PROGRAM PLC_AMX_AI
VAR_INPUT
	nSocketType:UINT:=1;// socket 类型; 0 表示 server; 1 表示 client;
	sTerminalName:STRING;// 通讯对方名称 自定义
	sHost:STRING(20):='127.0.0.1';// 通讯IP地址; server时表示本地host; client时表示远程host
	nPort:UDINT:=8900;// 通讯端口号;
	bEnable:BOOL:=TRUE;// 通讯启用\禁用连接
	sSendSuffix:STRING:='';//此处可统一添加发送后缀字符 $R$N
	nQueueInterval:UDINT:=50;// 发送队列时间间隔 单位ms
	logHandleArray:ARRAY [1..5] OF POINTER TO printLogModule_EX;// log 操作 handle 数组
	logHandleArrayLength:UINT:=0;// log 操作 handle 数组长度, 不超过5
	enHeartBeat:BOOL;// 启用心跳包命令
	cmdHeartBeat:DINT;// 心跳包命令
	readStateFlag:BOOL;
	volt:REAL;
	dworld:UDINT;
END_VAR
VAR_OUTPUT
	bSendCondition	:BOOL;//可发送条件
	bSocketConnected:BOOL;//连接状态
	
END_VAR
VAR CONSTANT
	cNumBegin		:DINT:=1;
	cNumEnd			:DINT:=100;
END_VAR
VAR
	sendDataArray	:ARRAY [cNumBegin..cNumEnd] OF struct_byte;
	length			:DINT:=0;
	endPoint		:DINT:=cNumBegin;
	sendPoint		:DINT:=cNumBegin;
	passMax			:BOOL;
	popupSendData	:struct_byte;
	//popup
	popupStep		:UINT:=0;
	popupTON1		:TON;
	popupTON2		:TON;
	iPopup			:DINT:=0;
	_PopupLength	:DINT:=0;
	sendDataTemp	:struct_byte;
	sendLenght		:UDINT;
END_VAR
VAR
	tcpipClient					:tcpipClientModule_EX;
	tcpipServer					:tcpipServerModule_EX;////定义服务器对象
	
	tcpipSendDataBuff_Server	:struct_byte;//发送数据 Buff server
	tcpipSendDataBuff_Client	:struct_byte;//发送数据 Buff client
	
	tcpipSendDataClear			:struct_byte;//发送数据 清空
	tcpipSendData				:struct_byte;//发送数据
	
	tcpipRecDataBuff_Server		:struct_byte;//已接收数据 Buff server
	tcpipRecDataBuff_Client		:struct_byte;//已接收数据 Buff client
	
	tcpipRecDataClear			:struct_byte;//已接收数据 清空
	tcpipRecData				:struct_byte;//已接收数据
	
	tcpConnectR_Trig			:R_Trig;//初始连接上升沿
	tcpConnectF_Trig			:F_Trig;//初始连接下降沿
	registerStep				:UDINT;//ALC注册控制步
	registerTON					:TON;//ALC注册延时
	
	logHandleArray_index		:UINT:=1;
	sendStep:UDINT;
	t1:TON;
	timeout1:TON;
	timeoutTimes:UDINT;
	disconnectedTon:TON;
END_VAR
VAR
	(*
	bTrig_Version:BOOL;
	rTrig_Version:R_TRIG;
	*)
END_VAR


CASE nSocketType OF
0://TCPIP server
	tcpipServer(
		sSrvNetId:= , 
		sLocalHost:=sHost , 
		nLocalPort:=nPort , 
		bStartConnect:=bEnable , 
		tcpipSDataLen:=sendLenght , 
		tcpipSData:=ADR(tcpipSendDataBuff_Server) , 
		bSend:= , 
		tcpipRecDataLen:=SIZEOF(tcpipRecDataBuff_Server), 
		tcpipRecData:=ADR(tcpipRecDataBuff_Server) , 
		bAccepted=> , 
		bSendBusy=> , 
		bRecData=> );
	bSendCondition:=tcpipServer.bAccepted AND NOT tcpipServer.bSendBusy;
	//TCPIP连接
	bSocketConnected:=tcpipServer.bAccepted;
	IF NOT tcpipServer.bAccepted THEN
		length:=0;
		endPoint:=cNumBegin;
		sendPoint:=cNumBegin;
		passMax:=FALSE;
	END_IF
	tcpConnectR_Trig(CLK:=tcpipServer.bAccepted);
	tcpConnectF_Trig(CLK:=tcpipServer.bAccepted);

1://TCPIP client
	tcpipClient(
		sSrvNetId:= , 
		sRemoteHost:=sHost , 
		nRemotePort:=nPort , 
		bStartConnect:=bEnable , 
		tcpipSDataLen:=sendLenght, 
		tcpipSData:=ADR(tcpipSendDataBuff_Client) , 
		bSend:= , 
		tcpipRecDataLen:=SIZEOF(tcpipRecDataBuff_Client) , 
		tcpipRecData:=ADR(tcpipRecDataBuff_Client) , 
		bConnected=> , 
		bSendBusy=> , 
		bRecData=> );
	bSendCondition:=tcpipClient.bConnected AND NOT tcpipClient.bSendBusy;
	//TCPIP连接
	bSocketConnected:=tcpipClient.bConnected;
	IF NOT tcpipClient.bConnected THEN
		length:=0;
		endPoint:=cNumBegin;
		sendPoint:=cNumBegin;
		passMax:=FALSE;
	END_IF
	tcpConnectR_Trig(CLK:=tcpipClient.bConnected);
	tcpConnectF_Trig(CLK:=tcpipClient.bConnected);
END_CASE

IF tcpConnectR_Trig.Q THEN
	FOR logHandleArray_index:=1 TO logHandleArrayLength DO
		logHandleArray[logHandleArray_index]^.append(CONCAT(sTerminalName, ' has been connected'));
	END_FOR
	registerStep:=10;
END_IF
IF tcpConnectF_Trig.Q THEN
	FOR logHandleArray_index:=1 TO logHandleArrayLength DO
		logHandleArray[logHandleArray_index]^.append(CONCAT(sTerminalName, ' has been disconnected'));
	END_FOR
	registerStep:=0;
END_IF
//数据接收处理
CASE nSocketType OF
0://TCPIP server
	IF tcpipServer.bRecData THEN
		tcpipRecData:=tcpipRecDataBuff_Server;//buff转存
		tcpipRecDataBuff_Server:=tcpipRecDataClear;//转存之后清空buff
		dataProcessing();
	END_IF
1://TCPIP client
	IF tcpipClient.bRecData THEN
		tcpipRecData:=tcpipRecDataBuff_Client;//buff转存
		tcpipRecDataBuff_Client:=tcpipRecDataClear;//转存之后清空buff
		dataProcessing();
	END_IF
END_CASE


popup();

CASE registerStep OF
0:
	//Ready
10:
	registerStep:=0;
// 心跳包
20:
	IF NOT enHeartBeat THEN
		registerStep:=0;
	ELSE
		registerStep:=registerStep+10;
	END_IF
30:
	registerTON(IN:=FALSE);
	registerStep:=registerStep+10;
40:
	registerTON(IN:=NOT registerTON.Q,PT:=T#3S);
	IF registerTON.Q THEN
		registerTON(IN:=FALSE);
		registerStep:=30;
	END_IF
END_CASE

CASE sendStep OF
0:
	sendStep:=10;
	timeout1(IN:=FALSE);
	t1(IN:=FALSE);
10:
	IF bSocketConnected THEN
		sendStep:=20;
	ELSE
		sendStep:=10;
	END_IF
// 心跳包
20:
	ReadVoltage();
	sendStep:=30;
30:
	IF readStateFlag THEN
		sendStep:=40;
		timeout1(IN:=FALSE);
		readStateFlag:=FALSE;
		timeoutTimes:=0;
		RETURN;
	END_IF
	timeout1(IN:=NOT timeout1.Q,PT:=T#1S);
	IF timeout1.Q THEN
		timeout1(IN:=FALSE);
		sendStep:=50;
		timeoutTimes:=timeoutTimes+1;
		IF timeoutTimes>3 THEN
			volt:=10.022;
			dworld:=4105;
			timeoutTimes:=0;
		END_IF
	END_IF
40:
	t1(IN:=NOT t1.Q,PT:=T#0.5S);
	IF t1.Q THEN
		t1(IN:=FALSE);
		sendStep:=50;
	END_IF
50:
	sendStep:=10;
END_CASE
disconnectedTon(IN:=NOT bSocketConnected,PT:=T#5S);
IF disconnectedTon.Q THEN
	volt:=10.022;
	dworld:=4105;
END_IF
Manual();

METHOD appendSend : BOOL
VAR_INPUT
	b1		:BYTE:=0;
	b2		:BYTE:=0;
	b3		:Byte:=0;
	b4		:Byte:=0;
	b5		:Byte:=0;
	b6		:Byte:=0;
	b7		:Byte:=0;
	b8		:Byte:=0;
	b9		:BYTE:=0;
	b10		:BYTE:=0;
	b11		:BYTE:=0;
	b12		:BYTE:=0;
	b13		:BYTE:=0;
	b14		:BYTE:=0;
	b15		:BYTE:=0;
	b16		:BYTE:=0;
	b17		:BYTE:=0;
	b18		:BYTE:=0;
	b19		:BYTE:=0;
	b20		:BYTE:=0;
	lenght	:UDINT;
END_VAR
sendLenght:=lenght;
sendDataArray[endPoint].b1:=b1;
sendDataArray[endPoint].b2:=b2;
sendDataArray[endPoint].b3:=b3;
sendDataArray[endPoint].b4:=b4;
sendDataArray[endPoint].b5:=b5;
sendDataArray[endPoint].b6:=b6;
sendDataArray[endPoint].b7:=b7;
sendDataArray[endPoint].b8:=b8;
sendDataArray[endPoint].b9:=b9;
sendDataArray[endPoint].b10:=b10;
sendDataArray[endPoint].b11:=b11;
sendDataArray[endPoint].b12:=b12;
sendDataArray[endPoint].b13:=b13;
sendDataArray[endPoint].b14:=b14;
sendDataArray[endPoint].b15:=b15;
sendDataArray[endPoint].b16:=b16;
sendDataArray[endPoint].b17:=b17;
sendDataArray[endPoint].b18:=b18;
sendDataArray[endPoint].b19:=b19;
sendDataArray[endPoint].b20:=b20;

endPoint:=endPoint+1;
IF endPoint>(cNumEnd-1) THEN
	endPoint:=1;
	passMax:=TRUE;
END_IF
END_METHOD

METHOD dataProcessing : BOOL
VAR_INPUT
END_VAR
VAR
	i_CGResult:INT;
	i_HResult:INT;
	str1:STRING;
END_VAR
FOR logHandleArray_index:=1 TO logHandleArrayLength DO
	CASE nSocketType OF
	0://TCPIP server
		str1:=CONCAT(str1,BYTE_TO_HEXSTR(tcpipRecData.b1,2,FALSE));
		str1:=CONCAT(str1,' ');
		str1:=CONCAT(str1,BYTE_TO_HEXSTR(tcpipRecData.b2,2,FALSE));
		str1:=CONCAT(str1,' ');
		str1:=CONCAT(str1,BYTE_TO_HEXSTR(tcpipRecData.b3,2,FALSE));
		str1:=CONCAT(str1,' ');
		str1:=CONCAT(str1,BYTE_TO_HEXSTR(tcpipRecData.b4,2,FALSE));
		str1:=CONCAT(str1,' ');
		str1:=CONCAT(str1,BYTE_TO_HEXSTR(tcpipRecData.b5,2,FALSE));
		str1:=CONCAT(str1,' ');
		str1:=CONCAT(str1,BYTE_TO_HEXSTR(tcpipRecData.b6,2,FALSE));
		str1:=CONCAT(str1,' ');
		str1:=CONCAT(str1,BYTE_TO_HEXSTR(tcpipRecData.b7,2,FALSE));
		str1:=CONCAT(str1,' ');
		str1:=CONCAT(str1,BYTE_TO_HEXSTR(tcpipRecData.b8,2,FALSE));
		str1:=CONCAT(str1,' ');
		str1:=CONCAT(str1,BYTE_TO_HEXSTR(tcpipRecData.b9,2,FALSE));
		str1:=CONCAT(str1,' ');
		str1:=CONCAT(str1,BYTE_TO_HEXSTR(tcpipRecData.b10,2,FALSE));
		str1:=CONCAT(str1,' ');
		str1:=CONCAT(str1,BYTE_TO_HEXSTR(tcpipRecData.b11,2,FALSE));
		str1:=CONCAT(str1,' ');
		str1:=CONCAT(str1,BYTE_TO_HEXSTR(tcpipRecData.b12,2,FALSE));
		str1:=CONCAT(str1,' ');
		str1:=CONCAT(str1,BYTE_TO_HEXSTR(tcpipRecData.b13,2,FALSE));
		str1:=CONCAT(str1,' ');
		str1:=CONCAT(str1,BYTE_TO_HEXSTR(tcpipRecData.b14,2,FALSE));
		str1:=CONCAT(str1,' ');
		str1:=CONCAT(str1,BYTE_TO_HEXSTR(tcpipRecData.b15,2,FALSE));
		str1:=CONCAT(str1,' ');
		str1:=CONCAT(str1,BYTE_TO_HEXSTR(tcpipRecData.b16,2,FALSE));
		str1:=CONCAT(str1,' ');
		str1:=CONCAT(str1,BYTE_TO_HEXSTR(tcpipRecData.b17,2,FALSE));
		str1:=CONCAT(str1,' ');
		str1:=CONCAT(str1,BYTE_TO_HEXSTR(tcpipRecData.b18,2,FALSE));
		str1:=CONCAT(str1,' ');
		str1:=CONCAT(str1,BYTE_TO_HEXSTR(tcpipRecData.b19,2,FALSE));
		str1:=CONCAT(str1,' ');
		str1:=CONCAT(str1,BYTE_TO_HEXSTR(tcpipRecData.b20,2,FALSE));
//		logHandleArray[logHandleArray_index]^.append(CONCAT(CONCAT(CONCAT('Recevie From ', sTerminalName), ' -- '),str1));
	1://TCPIP client
		str1:=CONCAT(str1,BYTE_TO_HEXSTR(tcpipRecData.b1,2,FALSE));
		str1:=CONCAT(str1,' ');
		str1:=CONCAT(str1,BYTE_TO_HEXSTR(tcpipRecData.b2,2,FALSE));
		str1:=CONCAT(str1,' ');
		str1:=CONCAT(str1,BYTE_TO_HEXSTR(tcpipRecData.b3,2,FALSE));
		str1:=CONCAT(str1,' ');
		str1:=CONCAT(str1,BYTE_TO_HEXSTR(tcpipRecData.b4,2,FALSE));
		str1:=CONCAT(str1,' ');
		str1:=CONCAT(str1,BYTE_TO_HEXSTR(tcpipRecData.b5,2,FALSE));
		str1:=CONCAT(str1,' ');
		str1:=CONCAT(str1,BYTE_TO_HEXSTR(tcpipRecData.b6,2,FALSE));
		str1:=CONCAT(str1,' ');
		str1:=CONCAT(str1,BYTE_TO_HEXSTR(tcpipRecData.b7,2,FALSE));
		str1:=CONCAT(str1,' ');
		str1:=CONCAT(str1,BYTE_TO_HEXSTR(tcpipRecData.b8,2,FALSE));
		str1:=CONCAT(str1,' ');
		str1:=CONCAT(str1,BYTE_TO_HEXSTR(tcpipRecData.b9,2,FALSE));
		str1:=CONCAT(str1,' ');
		str1:=CONCAT(str1,BYTE_TO_HEXSTR(tcpipRecData.b10,2,FALSE));
		str1:=CONCAT(str1,' ');
		str1:=CONCAT(str1,BYTE_TO_HEXSTR(tcpipRecData.b11,2,FALSE));
		str1:=CONCAT(str1,' ');
		str1:=CONCAT(str1,BYTE_TO_HEXSTR(tcpipRecData.b12,2,FALSE));
		str1:=CONCAT(str1,' ');
		str1:=CONCAT(str1,BYTE_TO_HEXSTR(tcpipRecData.b13,2,FALSE));
		str1:=CONCAT(str1,' ');
		str1:=CONCAT(str1,BYTE_TO_HEXSTR(tcpipRecData.b14,2,FALSE));
		str1:=CONCAT(str1,' ');
		str1:=CONCAT(str1,BYTE_TO_HEXSTR(tcpipRecData.b15,2,FALSE));
		str1:=CONCAT(str1,' ');
		str1:=CONCAT(str1,BYTE_TO_HEXSTR(tcpipRecData.b16,2,FALSE));
		str1:=CONCAT(str1,' ');
		str1:=CONCAT(str1,BYTE_TO_HEXSTR(tcpipRecData.b17,2,FALSE));
		str1:=CONCAT(str1,' ');
		str1:=CONCAT(str1,BYTE_TO_HEXSTR(tcpipRecData.b18,2,FALSE));
		str1:=CONCAT(str1,' ');
		str1:=CONCAT(str1,BYTE_TO_HEXSTR(tcpipRecData.b19,2,FALSE));
		str1:=CONCAT(str1,' ');
		str1:=CONCAT(str1,BYTE_TO_HEXSTR(tcpipRecData.b20,2,FALSE));
//		logHandleArray[logHandleArray_index]^.append(CONCAT(CONCAT(CONCAT('Recevie From ', sTerminalName), ' -- '),str1));
	END_CASE
END_FOR

// 数据处理
readStateFlag:=TRUE;
volt:=TO_REAL((tcpipRecData.b10*256+tcpipRecData.b11)/4096.0)*10.0;
dworld:=tcpipRecData.b10*256+tcpipRecData.b11;
END_METHOD

ACTION Manual:
(*
rTrig_Version(CLK:=bTrig_Version);
IF rTrig_Version.Q THEN
	appendSend(0,0,E_CmdID_SW.SW_GetVer,0.0,0.0,0.0,0.0,0.0,0,'');
END_IF
*)
END_ACTION

METHOD PRIVATE popup : BOOL
VAR_INPUT
END_VAR
CASE popupStep OF
0:
	IF (sendPoint<endPoint OR passMax) AND bSendCondition THEN
		popupSendData:=sendDataArray[sendPoint];
		sendData(popupSendData);//此处是调用信息发送
		popupStep:=10;
		sendPoint:=sendPoint+1;
		IF sendPoint>(cNumEnd-1) THEN
			sendPoint:=1;
			passMax:=FALSE;
		END_IF
	END_IF
10:
	popupTON2(IN:=NOT popupTON2.Q, PT:=T#2S);
	IF NOT bSendCondition OR popupTON2.Q THEN
		popupTON2(IN:=FALSE);
		popupStep:=11;
	END_IF
11:
	IF bSendCondition THEN
		popupStep:=12;
	END_IF
	popupTON1(IN:=FALSE);
12:
	//popupTON1(IN:=NOT popupTON1.Q,PT:=T#10MS);
	popupTON1(IN:=NOT popupTON1.Q,PT:=TO_TIME(nQueueInterval));
	IF popupTON1.Q THEN
		popupStep:=0;
	END_IF
END_CASE
END_METHOD

METHOD ReadVoltage : BOOL
VAR_INPUT
END_VAR
appendSend(16#00,16#00,16#00,16#00,16#00,16#06,16#01,16#04,16#00,16#00,16#00,16#04,0,0,0,0,0,0,0,0,12);// 读进电压字符串
END_METHOD

METHOD PRIVATE sendData : BOOL
VAR_INPUT
	dataStruct	:struct_byte;
END_VAR
VAR
	str1:STRING;
END_VAR
IF bSendCondition AND bEnable THEN
	tcpipSendData.b1	:=dataStruct.b1;
	tcpipSendData.b2	:=dataStruct.b2;
	tcpipSendData.b3	:=dataStruct.b3;
	tcpipSendData.b4	:=dataStruct.b4;
	tcpipSendData.b5	:=dataStruct.b5;
	tcpipSendData.b6	:=dataStruct.b6;
	tcpipSendData.b7	:=dataStruct.b7;
	tcpipSendData.b8	:=dataStruct.b8;
	tcpipSendData.b9	:=dataStruct.b9;
	tcpipSendData.b10	:=dataStruct.b10;
	tcpipSendData.b11	:=dataStruct.b11;
	tcpipSendData.b12	:=dataStruct.b12;
	tcpipSendData.b13	:=dataStruct.b13;
	tcpipSendData.b14	:=dataStruct.b14;
	tcpipSendData.b15	:=dataStruct.b15;
	tcpipSendData.b16	:=dataStruct.b16;
	tcpipSendData.b17	:=dataStruct.b17;
	tcpipSendData.b18	:=dataStruct.b18;
	tcpipSendData.b19	:=dataStruct.b19;
	tcpipSendData.b20	:=dataStruct.b20;
	
	CASE nSocketType OF
	0://TCPIP server
		tcpipSendDataBuff_Server:=tcpipSendData;
		tcpipSendData:=tcpipSendDataClear;	
		tcpipServer.bSend:=TRUE;
	1://TCPIP client
		tcpipSendDataBuff_Client:=tcpipSendData;
		tcpipSendData:=tcpipSendDataClear;	
		tcpipClient.bSend:=TRUE;
	END_CASE
	
	FOR logHandleArray_index:=1 TO logHandleArrayLength DO
		CASE nSocketType OF
		0://TCPIP server
			str1:=CONCAT(str1,BYTE_TO_HEXSTR(tcpipSendDataBuff_Server.b1,2,FALSE));
			str1:=CONCAT(str1,' ');
			str1:=CONCAT(str1,BYTE_TO_HEXSTR(tcpipSendDataBuff_Server.b2,2,FALSE));
			str1:=CONCAT(str1,' ');
			str1:=CONCAT(str1,BYTE_TO_HEXSTR(tcpipSendDataBuff_Server.b3,2,FALSE));
			str1:=CONCAT(str1,' ');
			str1:=CONCAT(str1,BYTE_TO_HEXSTR(tcpipSendDataBuff_Server.b4,2,FALSE));
			str1:=CONCAT(str1,' ');
			str1:=CONCAT(str1,BYTE_TO_HEXSTR(tcpipSendDataBuff_Server.b5,2,FALSE));
			str1:=CONCAT(str1,' ');
			str1:=CONCAT(str1,BYTE_TO_HEXSTR(tcpipSendDataBuff_Server.b6,2,FALSE));
			str1:=CONCAT(str1,' ');
			str1:=CONCAT(str1,BYTE_TO_HEXSTR(tcpipSendDataBuff_Server.b7,2,FALSE));
			str1:=CONCAT(str1,' ');
			str1:=CONCAT(str1,BYTE_TO_HEXSTR(tcpipSendDataBuff_Server.b8,2,FALSE));
			str1:=CONCAT(str1,' ');
			str1:=CONCAT(str1,BYTE_TO_HEXSTR(tcpipSendDataBuff_Server.b9,2,FALSE));
			str1:=CONCAT(str1,' ');
			str1:=CONCAT(str1,BYTE_TO_HEXSTR(tcpipSendDataBuff_Server.b10,2,FALSE));
			str1:=CONCAT(str1,' ');
			str1:=CONCAT(str1,BYTE_TO_HEXSTR(tcpipSendDataBuff_Server.b11,2,FALSE));
			str1:=CONCAT(str1,' ');
			str1:=CONCAT(str1,BYTE_TO_HEXSTR(tcpipSendDataBuff_Server.b12,2,FALSE));
			str1:=CONCAT(str1,' ');
			str1:=CONCAT(str1,BYTE_TO_HEXSTR(tcpipSendDataBuff_Server.b13,2,FALSE));
			str1:=CONCAT(str1,' ');
			str1:=CONCAT(str1,BYTE_TO_HEXSTR(tcpipSendDataBuff_Server.b14,2,FALSE));
			str1:=CONCAT(str1,' ');
			str1:=CONCAT(str1,BYTE_TO_HEXSTR(tcpipSendDataBuff_Server.b15,2,FALSE));
			str1:=CONCAT(str1,' ');
			str1:=CONCAT(str1,BYTE_TO_HEXSTR(tcpipSendDataBuff_Server.b16,2,FALSE));
			str1:=CONCAT(str1,' ');
			str1:=CONCAT(str1,BYTE_TO_HEXSTR(tcpipSendDataBuff_Server.b17,2,FALSE));
			str1:=CONCAT(str1,' ');
			str1:=CONCAT(str1,BYTE_TO_HEXSTR(tcpipSendDataBuff_Server.b18,2,FALSE));
			str1:=CONCAT(str1,' ');
			str1:=CONCAT(str1,BYTE_TO_HEXSTR(tcpipSendDataBuff_Server.b19,2,FALSE));
			str1:=CONCAT(str1,' ');
			str1:=CONCAT(str1,BYTE_TO_HEXSTR(tcpipSendDataBuff_Server.b20,2,FALSE));
//			logHandleArray[logHandleArray_index]^.append(CONCAT(CONCAT(CONCAT('Send To ', sTerminalName), ' -- '),str1));
		1://TCPIP client
			str1:=CONCAT(str1,' ');
			str1:=CONCAT(str1,BYTE_TO_HEXSTR(tcpipSendDataBuff_Client.b1,2,FALSE));
			str1:=CONCAT(str1,' ');
			str1:=CONCAT(str1,BYTE_TO_HEXSTR(tcpipSendDataBuff_Client.b2,2,FALSE));
			str1:=CONCAT(str1,' ');
			str1:=CONCAT(str1,BYTE_TO_HEXSTR(tcpipSendDataBuff_Client.b3,2,FALSE));
			str1:=CONCAT(str1,' ');
			str1:=CONCAT(str1,BYTE_TO_HEXSTR(tcpipSendDataBuff_Client.b4,2,FALSE));
			str1:=CONCAT(str1,' ');
			str1:=CONCAT(str1,BYTE_TO_HEXSTR(tcpipSendDataBuff_Client.b5,2,FALSE));
			str1:=CONCAT(str1,' ');
			str1:=CONCAT(str1,BYTE_TO_HEXSTR(tcpipSendDataBuff_Client.b6,2,FALSE));
			str1:=CONCAT(str1,' ');
			str1:=CONCAT(str1,BYTE_TO_HEXSTR(tcpipSendDataBuff_Client.b7,2,FALSE));
			str1:=CONCAT(str1,' ');
			str1:=CONCAT(str1,BYTE_TO_HEXSTR(tcpipSendDataBuff_Client.b8,2,FALSE));
			str1:=CONCAT(str1,' ');
			str1:=CONCAT(str1,BYTE_TO_HEXSTR(tcpipSendDataBuff_Client.b9,2,FALSE));
			str1:=CONCAT(str1,' ');
			str1:=CONCAT(str1,BYTE_TO_HEXSTR(tcpipSendDataBuff_Client.b10,2,FALSE));
			str1:=CONCAT(str1,' ');
			str1:=CONCAT(str1,BYTE_TO_HEXSTR(tcpipSendDataBuff_Client.b11,2,FALSE));
			str1:=CONCAT(str1,' ');
			str1:=CONCAT(str1,BYTE_TO_HEXSTR(tcpipSendDataBuff_Client.b12,2,FALSE));
			str1:=CONCAT(str1,' ');
			str1:=CONCAT(str1,BYTE_TO_HEXSTR(tcpipSendDataBuff_Client.b13,2,FALSE));
			str1:=CONCAT(str1,' ');
			str1:=CONCAT(str1,BYTE_TO_HEXSTR(tcpipSendDataBuff_Client.b14,2,FALSE));
			str1:=CONCAT(str1,' ');
			str1:=CONCAT(str1,BYTE_TO_HEXSTR(tcpipSendDataBuff_Client.b15,2,FALSE));
			str1:=CONCAT(str1,' ');
			str1:=CONCAT(str1,BYTE_TO_HEXSTR(tcpipSendDataBuff_Client.b16,2,FALSE));
			str1:=CONCAT(str1,' ');
			str1:=CONCAT(str1,BYTE_TO_HEXSTR(tcpipSendDataBuff_Client.b17,2,FALSE));
			str1:=CONCAT(str1,' ');
			str1:=CONCAT(str1,BYTE_TO_HEXSTR(tcpipSendDataBuff_Client.b18,2,FALSE));
			str1:=CONCAT(str1,' ');
			str1:=CONCAT(str1,BYTE_TO_HEXSTR(tcpipSendDataBuff_Client.b19,2,FALSE));
			str1:=CONCAT(str1,' ');
			str1:=CONCAT(str1,BYTE_TO_HEXSTR(tcpipSendDataBuff_Client.b20,2,FALSE));
//			logHandleArray[logHandleArray_index]^.append(CONCAT(CONCAT(CONCAT('Send To ', sTerminalName), ' -- '),str1));
		END_CASE
	END_FOR
END_IF
END_METHOD

END_PROGRAM

(* stored: Version 1.1.0.1, ProductVersion 3.1.4024.12
   POU PLC_AMX_AI: Id {39e2c8be-759d-4f9b-8129-7a38178d708d}, SpecialFunc None
   Folder CMD: Id {425ceb4c-30b5-43e8-b60b-b054739507e2}
   Folder Recevie: Id {aea389ea-09ce-4eb8-997c-367412738621}
   Folder Send: Id {dc9c1c98-59e9-4575-93b5-03320632d237}
   Folder Private: Id {316b3631-165e-4dea-af61-bbc66624c62f}
   Method appendSend: Id {0ce465e2-e0e9-4392-822e-5e85489ce395}
   Method dataProcessing: Id {41b6ac29-656e-470e-856e-7a0383710dcd}
   Action Manual: Id {18d5dfc7-12da-4a5c-9a7d-d74222d8711c}
   Method popup: Id {c931ef7c-fa0b-413e-96d6-8e5422f72068}
   Method ReadVoltage: Id {93a31dd3-5c13-47d5-8df5-57865b48c963}
   Method sendData: Id {00f63878-d5fb-484c-859f-c9ae840c0f9a} *)
